Fanuc KAREL source: kt00029.KL

-- PROVISIONAL review KL for V770-1; original PC SHA256 3076aade4059a7030f9a7cba5021952de4ae98b438a42a14f07eed44ea1390c2
-- Incomplete behavior may be omitted. Consult companion uncertainty JSON. Do not deploy.
PROGRAM KT00029
%NOLOCKGROUP
VAR
  OUT : INTEGER
-- UNRESOLVED_DECL H1 type=002017
-- UNRESOLVED_DECL Y2 type=002018
BEGIN
  -- UNRESOLVED_PC offsets 5-19; opcodes 2E,22,9D,33,B4
  -- UNRESOLVED_PC offsets 24-38; opcodes 2E,22,9D,33,B2
  -- UNRESOLVED_PC offsets 43-68; opcodes 22,9D,33,B3,22,9D,33,B1,52,23
  -- UNRESOLVED_PC offsets 73-77; opcodes 7F
END KT00029
